PROGRAM PRG_TEST
VAR
	fbRunHOMSTest : FB_RunHOMS_Test;
END_VAR

TcUnit.RUN();

END_PROGRAM

(* stored: Version 1.1.0.1, ProductVersion 3.1.4024.3
   POU PRG_TEST: Id {c9df370d-c0ed-441f-b0c3-9ace7414a6e0}, SpecialFunc None *)
